// TIA Portal V15.1 export
// export: Created 2024-06-21T08:40:53.4911865Z, ExportSetting WithDefaults, DisplayName Totally Integrated Automation Portal, DisplayVersion V15.1 Update 5, DisplayName TIA Portal Openness, DisplayVersion V15.1 Update 5, DisplayName SINAMICS Startdrive Advanced, DisplayVersion V15.1, DisplayName G130, G150, S120, S150, SINAMICS MV, S210, DisplayVersion V15.1, DisplayName G110M, G120, G120C, G120D, G120P, DisplayVersion V15.1, DisplayName STEP 7 Professional, DisplayVersion V15.1 Update 5, DisplayName STEP 7 Safety, DisplayVersion V15.1, DisplayName WinCC Professional, DisplayVersion V15.1 Update 5, DisplayName SIMATIC Visualization Architect, DisplayVersion V15.1
FUNCTION "LIAnimDWord" : Void   // FC1005, FBD
TITLE = LIAnimDWord
{ S7_Optimized_Access := 'TRUE' }
AUTHOR : VCC
FAMILY : Anim
NAME : SIAnim
VERSION : 0.1
// =============================================================================
// Handles the conversion from bits to one Word for simple icon Animation. 
// =============================================================================
// stored: AutoNumber false, IsIECCheckEnabled false, SetENOAutomatically False, UDAEnableTagReadback false
   VAR_INPUT
      I_SetPos : Bool;   // Set position / Set Position
      I_ResetPos : Bool;   // Reset position / Reset Position
      I_Active : Bool;   // Active
      I_Visible : Bool;   // ObjectVisible
      I_OutOfUse : Bool;   // Object out of use
      I_IntlkSet : Bool;   // Interlock for Set direction
      I_IntlkReset : Bool;   // Interlock for Reset direction
      I_IntlkSetAlm : Bool;   // Interlock alarm for Set direction / Interlock Alarm for Set direction
      I_IntlkResetAlm : Bool;   // Interlock alarm for Reset direction / Interlock Alarm for Reset direction
      I_ManualMode : Bool;   // Manual mode / Manual Mode
      I_FncSelInHMI : Bool;   // Manual selection from HMI
      I_AnySelected : Bool;   // Something is Selected
      I_AlarmA : Bool;   // AlarmA
      I_AlarmB : Bool;   // AlarmB
      I_AlarmC : Bool;   // AlarmC
      I_AlarmD : Bool;   // AlarmD
      I_SafetyOk : Bool;   // Safety Ok
      I_Service : Bool;   // Service Active
      I_Spare1 : Bool;   // Spare
      I_Spare2 : Bool;   // Spare
      I_Spare3 : Bool;   // Spare
      I_Spare4 : Bool;   // Spare
      I_Spare5 : Bool;   // Spare
      I_Spare6 : Bool;   // Spare
      I_Spare7 : Bool;   // Spare
      I_Spare8 : Bool;   // Spare
      I_Spare9 : Bool;   // Spare
      I_Spare10 : Bool;   // Spare
      I_Spare11 : Bool;   // Spare
      I_Spare12 : Bool;   // Spare
      I_Spare13 : Bool;   // Spare
      I_Spare14 : Bool;   // Spare
   END_VAR
   VAR_OUTPUT
      H_IAnim : DWord;   // Icon animation Word / Icon Animation
   END_VAR
BEGIN

REGION Network 1: Icon animation Word / **** 1 - Inputs **** Set position
   // Set Position
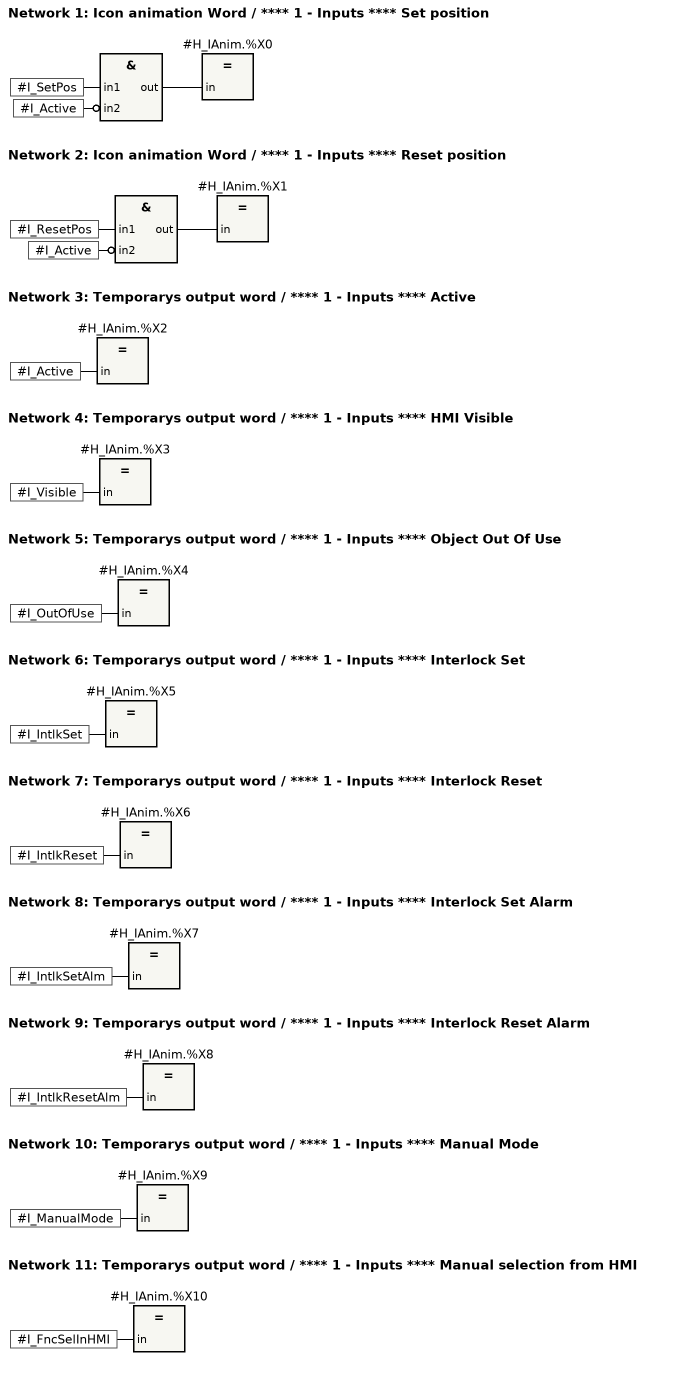
   #H_IAnim.%X0 := #I_SetPos AND NOT #I_Active;
END_REGION

REGION Network 2: Icon animation Word / **** 1 - Inputs **** Reset position
   // Reset Position
   #H_IAnim.%X1 := #I_ResetPos AND NOT #I_Active;
END_REGION

REGION Network 3: Temporarys output word / **** 1 - Inputs **** Active
   // Active
   #H_IAnim.%X2 := #I_Active;
END_REGION

REGION Network 4: Temporarys output word / **** 1 - Inputs **** HMI Visible
   // HMI Visible
   #H_IAnim.%X3 := #I_Visible;
END_REGION

REGION Network 5: Temporarys output word / **** 1 - Inputs **** Object Out Of Use
   // Object out of use
   #H_IAnim.%X4 := #I_OutOfUse;
END_REGION

REGION Network 6: Temporarys output word / **** 1 - Inputs **** Interlock Set
   // Interlock Set
   #H_IAnim.%X5 := #I_IntlkSet;
END_REGION

REGION Network 7: Temporarys output word / **** 1 - Inputs **** Interlock Reset
   // Interlock Reset
   #H_IAnim.%X6 := #I_IntlkReset;
END_REGION

REGION Network 8: Temporarys output word / **** 1 - Inputs **** Interlock Set Alarm
   // Interlock Set Alarm
   #H_IAnim.%X7 := #I_IntlkSetAlm;
END_REGION

REGION Network 9: Temporarys output word / **** 1 - Inputs **** Interlock Reset Alarm
   // Interlock Reset Alarm
   #H_IAnim.%X8 := #I_IntlkResetAlm;
END_REGION

REGION Network 10: Temporarys output word / **** 1 - Inputs **** Manual Mode
   // Manual Mode
   #H_IAnim.%X9 := #I_ManualMode;
END_REGION

REGION Network 11: Temporarys output word / **** 1 - Inputs **** Manual selection from HMI
   // Manual selection from HMI
   #H_IAnim.%X10 := #I_FncSelInHMI;
END_REGION

REGION Network 12: Temporarys output word / **** 1 - Inputs **** Selected
   // Selected
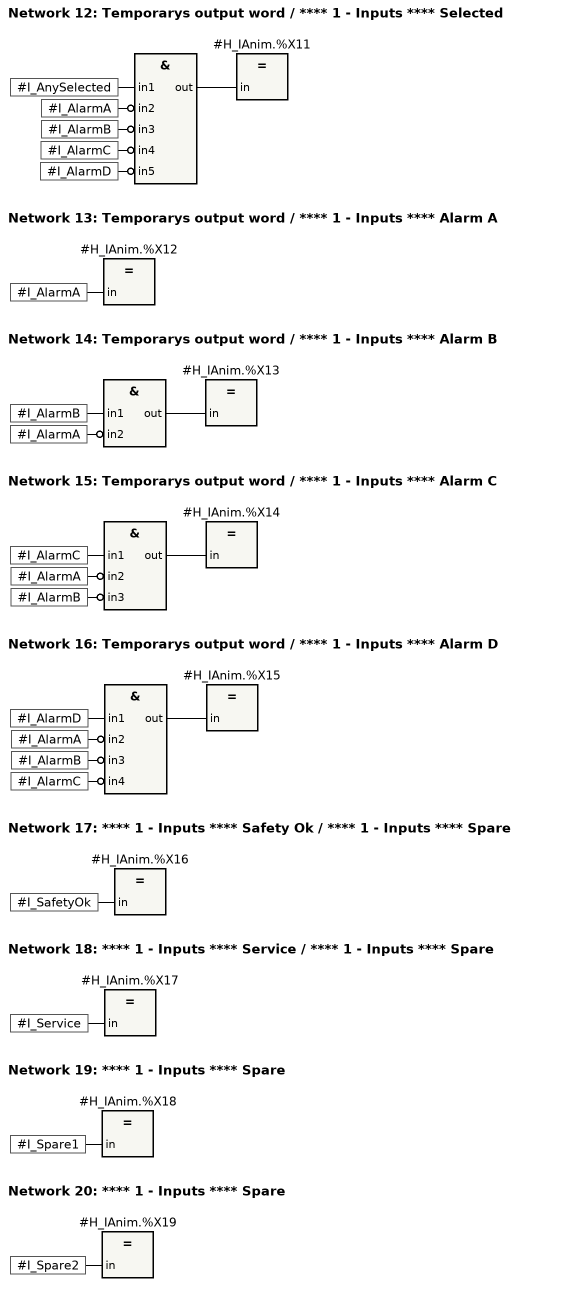
   #H_IAnim.%X11 := #I_AnySelected AND NOT #I_AlarmA AND NOT #I_AlarmB AND NOT #I_AlarmC AND NOT #I_AlarmD;
END_REGION

REGION Network 13: Temporarys output word / **** 1 - Inputs **** Alarm A
   // Alarm A
   #H_IAnim.%X12 := #I_AlarmA;
END_REGION

REGION Network 14: Temporarys output word / **** 1 - Inputs **** Alarm B
   // Alarm B
   #H_IAnim.%X13 := #I_AlarmB AND NOT #I_AlarmA;
END_REGION

REGION Network 15: Temporarys output word / **** 1 - Inputs **** Alarm C
   // Alarm C
   #H_IAnim.%X14 := #I_AlarmC AND NOT #I_AlarmA AND NOT #I_AlarmB;
END_REGION

REGION Network 16: Temporarys output word / **** 1 - Inputs **** Alarm D
   // Alarm D
   #H_IAnim.%X15 := #I_AlarmD AND NOT #I_AlarmA AND NOT #I_AlarmB AND NOT #I_AlarmC;
END_REGION

REGION Network 17: **** 1 - Inputs **** Safety Ok / **** 1 - Inputs **** Spare
   // Safety Ok / Spare
   #H_IAnim.%X16 := #I_SafetyOk;
END_REGION

REGION Network 18: **** 1 - Inputs **** Service / **** 1 - Inputs **** Spare
   // Service / Spare
   #H_IAnim.%X17 := #I_Service;
END_REGION

REGION Network 19: **** 1 - Inputs **** Spare
   // Spare
   #H_IAnim.%X18 := #I_Spare1;
END_REGION

REGION Network 20: **** 1 - Inputs **** Spare
   // Spare
   #H_IAnim.%X19 := #I_Spare2;
END_REGION

REGION Network 21: **** 1 - Inputs **** Spare
   // Spare
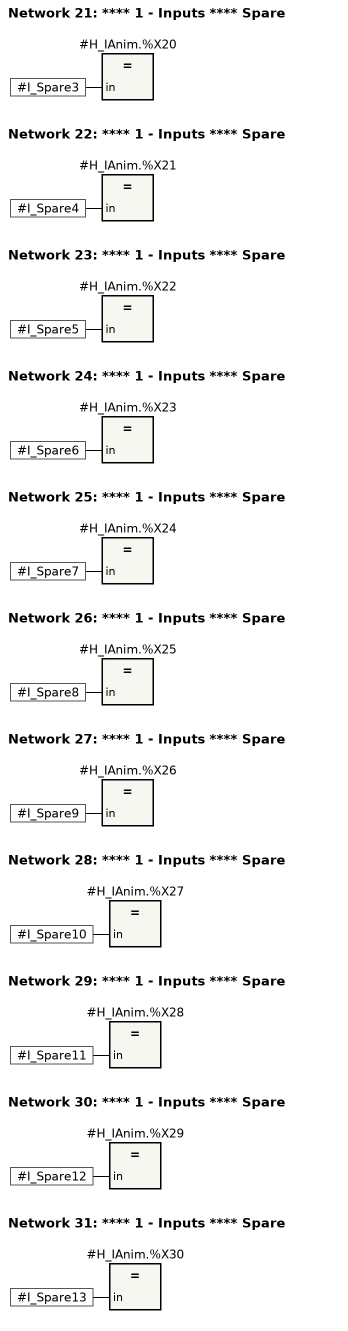
   #H_IAnim.%X20 := #I_Spare3;
END_REGION

REGION Network 22: **** 1 - Inputs **** Spare
   // Spare
   #H_IAnim.%X21 := #I_Spare4;
END_REGION

REGION Network 23: **** 1 - Inputs **** Spare
   // Spare
   #H_IAnim.%X22 := #I_Spare5;
END_REGION

REGION Network 24: **** 1 - Inputs **** Spare
   // Spare
   #H_IAnim.%X23 := #I_Spare6;
END_REGION

REGION Network 25: **** 1 - Inputs **** Spare
   // Spare
   #H_IAnim.%X24 := #I_Spare7;
END_REGION

REGION Network 26: **** 1 - Inputs **** Spare
   // Spare
   #H_IAnim.%X25 := #I_Spare8;
END_REGION

REGION Network 27: **** 1 - Inputs **** Spare
   // Spare
   #H_IAnim.%X26 := #I_Spare9;
END_REGION

REGION Network 28: **** 1 - Inputs **** Spare
   // Spare
   #H_IAnim.%X27 := #I_Spare10;
END_REGION

REGION Network 29: **** 1 - Inputs **** Spare
   // Spare
   #H_IAnim.%X28 := #I_Spare11;
END_REGION

REGION Network 30: **** 1 - Inputs **** Spare
   // Spare
   #H_IAnim.%X29 := #I_Spare12;
END_REGION

REGION Network 31: **** 1 - Inputs **** Spare
   // Spare
   #H_IAnim.%X30 := #I_Spare13;
END_REGION

REGION Network 32: **** 1 - Inputs **** Spare
   // Spare
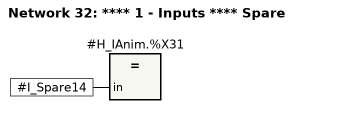
   #H_IAnim.%X31 := #I_Spare14;
END_REGION
END_FUNCTION
